TYPE hmiCommandsJog_TypeStruct :
STRUCT
		
	jogFw	 :BOOL;
	jogRev	: BOOL;

END_STRUCT
END_TYPE

(* stored: Version 1.1.0.1
   DUT hmiCommandsJog_TypeStruct: Id {343b7bfb-5cb4-4457-8791-48f3d2005ef9} *)
